{attribute addProperty BoxType "EL5101-0000-1020"}
{attribute addProperty Id "Latch_C_validBIT10.1251Latch_extern_validBIT10.1252Set_counter_doneBIT10.1253Counter_underflowBIT10.1254Counter_overflowBIT10.1255Status_of_input_statusBIT10.1256Open_circuitBIT10.1257Extrapolation_stallBIT10.1258Status_of_input_ABIT10.1259Status_of_input_BBIT10.12510Status_of_input_CBIT10.12511Status_of_input_gateBIT10.12512Status_of_extern_latchBIT10.12513Sync_ErrorBIT10.12532TxPDO_StateBIT10.1257TxPDO_ToggleBIT10.1259"}
{attribute addProperty CRC "3131182327"}
{attribute addProperty SizeInBites "16"}
{attribute addProperty SizeInBytes "2"}
TYPE Status_BAA20CF7 :
STRUCT
	{attribute addProperty Name "Latch_C_valid"}
	Latch_C_valid : BIT;
	{attribute addProperty Name "Latch_extern_valid"}
	Latch_extern_valid : BIT;
	{attribute addProperty Name "Set_counter_done"}
	Set_counter_done : BIT;
	{attribute addProperty Name "Counter_underflow"}
	Counter_underflow : BIT;
	{attribute addProperty Name "Counter_overflow"}
	Counter_overflow : BIT;
	{attribute addProperty Name "Status_of_input_status"}
	Status_of_input_status : BIT;
	{attribute addProperty Name "Open_circuit"}
	Open_circuit : BIT;
	{attribute addProperty Name "Extrapolation_stall"}
	Extrapolation_stall : BIT;
	{attribute addProperty Name "Status_of_input_A"}
	Status_of_input_A : BIT;
	{attribute addProperty Name "Status_of_input_B"}
	Status_of_input_B : BIT;
	{attribute addProperty Name "Status_of_input_C"}
	Status_of_input_C : BIT;
	{attribute addProperty Name "Status_of_input_gate"}
	Status_of_input_gate : BIT;
	{attribute addProperty Name "Status_of_extern_latch"}
	Status_of_extern_latch : BIT;
	{attribute addProperty Name "Sync_Error"}
	Sync_Error : BIT;
	{attribute addProperty Name "TxPDO_State"}
	TxPDO_State : BIT;
	{attribute addProperty Name "TxPDO_Toggle"}
	TxPDO_Toggle : BIT;
END_STRUCT
END_TYPE

(* stored: Version 1.2.0.0, ProductVersion 3.1.4024.9
   DUT Status_BAA20CF7: Id {ac0ec866-545b-4115-9dc5-9b26cd7f2cff} *)
